(* IEC 61131-3 sources: RL_MAR/experiments/comparison/llm4plc/results/gpt-4o_20260507_114630/20260507_114736, 2 files *)

(* ---- generated_code_iteration_0.st ---- *)
plaintext
START_ST
FUNCTION_BLOCK FB_CalculateDayOfYear
VAR_INPUT
    Year: INT; // Input year (valid range: 1000-3000)
    Month: INT; // Input month (valid range: 1-12)
    Day: INT; // Input day (valid range depends on month and leap year)
END_VAR

VAR_OUTPUT
    DayOfYear: INT; // Output day of the year (1-366)
    error: BOOL; // Error flag
    status: WORD; // Error status code
END_VAR

VAR
    DaysInMonth: ARRAY[1..12] OF INT := [31, 28, 31, 30, 31, 30, 31, 31, 30, 31, 30, 31]; // Standard days in each month
    isLeapYear: BOOL; // Flag to indicate if the year is a leap year
    sumDays: INT; // Accumulator for summing days in completed months
    state: INT; // State variable to track the FSM state
END_VAR

// Main logic
CASE state OF

    // STATE 0: INITIALIZE
    0:
        DayOfYear := 0;
        error := FALSE;
        status := 0;
        isLeapYear := FALSE;
        sumDays := 0;
        state := 1; // Transition to STATE 1: VALIDATE MONTH

    // STATE 1: VALIDATE MONTH
    1:
        IF Month < 1 OR Month > 12 THEN
            error := TRUE;
            status := 16#8002; // Invalid month
            state := 5; // Transition to STATE 5: OUTPUT RESULTS
        ELSE
            state := 2; // Transition to STATE 2: VALIDATE YEAR
        END_IF;

    // STATE 2: VALIDATE YEAR
    2:
        IF Year < 1000 OR Year > 3000 THEN
            error := TRUE;
            status := 16#8001; // Invalid year
            state := 5; // Transition to STATE 5: OUTPUT RESULTS
        ELSE
            // Determine if the year is a leap year
            isLeapYear := (Year MOD 4 = 0 AND Year MOD 100 <> 0) OR (Year MOD 400 = 0);
            IF isLeapYear THEN
                DaysInMonth[2] := 29; // Adjust February days for leap year
            ELSE
                DaysInMonth[2] := 28; // Standard February days
            END_IF;
            state := 3; // Transition to STATE 3: VALIDATE DAY
        END_IF;

    // STATE 3: VALIDATE DAY
    3:
        IF Day <= 0 OR Day > DaysInMonth[Month] THEN
            error := TRUE;
            status := 16#8003; // Invalid day
            state := 5; // Transition to STATE 5: OUTPUT RESULTS
        ELSE
            state := 4; // Transition to STATE 4: CALCULATE DAY OF YEAR
        END_IF;

    // STATE 4: CALCULATE DAY OF YEAR
    4:
        sumDays := 0;
        FOR i := 1 TO Month - 1 DO
            sumDays := sumDays + DaysInMonth[i]; // Sum days of completed months
        END_FOR;
        DayOfYear := sumDays + Day; // Add the current day
        state := 5; // Transition to STATE 5: OUTPUT RESULTS

    // STATE 5: OUTPUT RESULTS
    5:
        IF NOT error THEN
            status := 0; // Success
        END_IF;
        state := 0; // Reset state to INITIALIZE for next execution

END_CASE;
END_FUNCTION_BLOCK
END_ST

(* ---- generated_code_iteration_1.st ---- *)
START_REASON
The error reported by the CODESYS compiler indicates that the identifier `i` was not defined in the `FOR` loop within the `STATE 4: CALCULATE DAY OF YEAR` section of the code. This issue occurred because the variable `i` was used in the loop without being declared in the `VAR` section. In Structured Text (ST), all variables must be explicitly declared before use. To fix this issue, the variable `i` needs to be added to the `VAR` section as an integer. Once this is done, the code should compile and function correctly.
END_REASON

START_ST
FUNCTION_BLOCK FB_CalculateDayOfYear
VAR_INPUT
    Year: INT; // Input year (valid range: 1000-3000)
    Month: INT; // Input month (valid range: 1-12)
    Day: INT; // Input day (valid range depends on month and leap year)
END_VAR

VAR_OUTPUT
    DayOfYear: INT; // Output day of the year (1-366)
    error: BOOL; // Error flag
    status: WORD; // Error status code
END_VAR

VAR
    DaysInMonth: ARRAY[1..12] OF INT := [31, 28, 31, 30, 31, 30, 31, 31, 30, 31, 30, 31]; // Standard days in each month
    isLeapYear: BOOL; // Flag to indicate if the year is a leap year
    sumDays: INT; // Accumulator for summing days in completed months
    state: INT; // State variable to track the FSM state
    i: INT; // Loop variable for iterating through months
END_VAR

// Main logic
CASE state OF

    // STATE 0: INITIALIZE
    0:
        DayOfYear := 0;
        error := FALSE;
        status := 0;
        isLeapYear := FALSE;
        sumDays := 0;
        state := 1; // Transition to STATE 1: VALIDATE MONTH

    // STATE 1: VALIDATE MONTH
    1:
        IF Month < 1 OR Month > 12 THEN
            error := TRUE;
            status := 16#8002; // Invalid month
            state := 5; // Transition to STATE 5: OUTPUT RESULTS
        ELSE
            state := 2; // Transition to STATE 2: VALIDATE YEAR
        END_IF;

    // STATE 2: VALIDATE YEAR
    2:
        IF Year < 1000 OR Year > 3000 THEN
            error := TRUE;
            status := 16#8001; // Invalid year
            state := 5; // Transition to STATE 5: OUTPUT RESULTS
        ELSE
            // Determine if the year is a leap year
            isLeapYear := (Year MOD 4 = 0 AND Year MOD 100 <> 0) OR (Year MOD 400 = 0);
            IF isLeapYear THEN
                DaysInMonth[2] := 29; // Adjust February days for leap year
            ELSE
                DaysInMonth[2] := 28; // Standard February days
            END_IF;
            state := 3; // Transition to STATE 3: VALIDATE DAY
        END_IF;

    // STATE 3: VALIDATE DAY
    3:
        IF Day <= 0 OR Day > DaysInMonth[Month] THEN
            error := TRUE;
            status := 16#8003; // Invalid day
            state := 5; // Transition to STATE 5: OUTPUT RESULTS
        ELSE
            state := 4; // Transition to STATE 4: CALCULATE DAY OF YEAR
        END_IF;

    // STATE 4: CALCULATE DAY OF YEAR
    4:
        sumDays := 0;
        FOR i := 1 TO Month - 1 DO
            sumDays := sumDays + DaysInMonth[i]; // Sum days of completed months
        END_FOR;
        DayOfYear := sumDays + Day; // Add the current day
        state := 5; // Transition to STATE 5: OUTPUT RESULTS

    // STATE 5: OUTPUT RESULTS
    5:
        IF NOT error THEN
            status := 0; // Success
        END_IF;
        state := 0; // Reset state to INITIALIZE for next execution

END_CASE;
END_FUNCTION_BLOCK
END_ST
